Fanuc TP program (LS listing): _Z_TEST_PLUGIN.LS

/PROG  _Z_TEST_PLUGIN
/ATTR
OWNER		= MNEDITOR;
COMMENT		= "";
PROG_SIZE	= 268;
CREATE		= DATE 22-07-02  TIME 21:53:28;
MODIFIED	= DATE 22-07-02  TIME 22:19:58;
FILE_NAME	= ;
VERSION		= 0;
LINE_COUNT	= 3;
MEMORY_SIZE	= 636;
PROTECT		= READ_WRITE;
TCD:  STACK_SIZE	= 0,
      TASK_PRIORITY	= 50,
      TIME_SLICE	= 0,
      BUSY_LAMP_OFF	= 0,
      ABORT_REQUEST	= 0,
      PAUSE_REQUEST	= 0;
DEFAULT_GROUP	= 1,*,*,*,*;
CONTROL_CODE	= 00000000 00000000;
LOCAL_REGISTERS	= 1,0,1;
/APPL

AUTO_SINGULARITY_HEADER;
  ENABLE_SINGULARITY_AVOIDANCE   : FALSE;
  ARC Welding Equipment : 1,*,*,*,*;
/MN
   1:  CALL IPL_FANUC_SWELD_SET(1,2,10,3,1,25,'_Z_GEN_SWELD') ;
   2: ;
   2:   R[10001]=$[IPL_FANUC_SWELD_CFG]KLSTAT ;
   2:   SR[10001]=$[IPL_FANUC_SWELD_CFG]TP_NAME ;
   3:  CALL SR[25]    ;
/POS
/END
